TYPE ST_PneumaticAxisOutputs :
STRUCT
    bSolenoid1On AT %Q*: BOOL; //Output of the solenoid valve 1
    bSolenoid2On AT %Q*: BOOL; //Output of the solenoid valve 2
END_STRUCT
END_TYPE

(* stored: Version 1.1.0.1
   DUT ST_PneumaticAxisOutputs: Id {aac9e877-b6e0-0811-2196-0106181b1955} *)
